PROGRAM MAIN
VAR	
	generateRecipe : BOOL;
	
	addRecipeToDB : AddRecipeToDatabase;
	validator : Validation;
	arrayHelpers : ArrayFunctions;
	
	resetAddRecipeToDatabase : AddRecipeToDatabase;
	resetValidation : Validation;
	resetArrayFunctions : ArrayFunctions;
	
	start : BOOL := TRUE;
END_VAR

validator(); //real time error/warning message generator

IF generateRecipe THEN
	addRecipeToDB();
	
	IF addRecipeToDB.finished THEN
		reset();
		//reset all variables
		generateRecipe := FALSE;
		RETURN;
	END_IF
END_IF

METHOD reset : BOOL
VAR_INPUT
END_VAR
//reset FBs
MEMCPY(ADR(addRecipeToDB), ADR(resetAddRecipeToDatabase), SIZEOF(AddRecipeToDatabase));
MEMCPY(ADR(validator), ADR(resetValidation), SIZEOF(Validation));
MEMCPY(ADR(arrayHelpers), ADR(resetArrayFunctions), SIZEOF(ArrayFunctions));

//reset fields
BundleData.id := '';
BundleData.weight := 0;
BundleData.length := 0;
BundleData.height := 0;
BundleData.width := 0;
BundleData.pieces := 0;
BundleData.layers := 0;
BundleData.piecesPerLayer := 0;
MEMSET(ADR(BundleData.requiredProcessing), 0, SIZEOF(BundleData.requiredProcessing));

ExtrusionData.extrusionWeight := 0;
ExtrusionData.extrusionHeight := 0;
ExtrusionData.extrusionWidth := 0;

MEMSET(ADR(StrapWrapRecipe.facePaper), 0, SIZEOF(StrapWrapRecipe.facePaper));
MEMSET(ADR(StrapWrapRecipe.faceCardboard), 0, SIZEOF(StrapWrapRecipe.faceCardboard));
MEMSET(ADR(StrapWrapRecipe.TopPaper), 0, SIZEOF(StrapWrapRecipe.TopPaper));
MEMSET(ADR(StrapWrapRecipe.LeftPaper), 0, SIZEOF(StrapWrapRecipe.LeftPaper));
MEMSET(ADR(StrapWrapRecipe.RightPaper), 0, SIZEOF(StrapWrapRecipe.RightPaper));
MEMSET(ADR(StrapWrapRecipe.BottomPaper), 0, SIZEOF(StrapWrapRecipe.BottomPaper));
MEMSET(ADR(StrapWrapRecipe.Cardboard), 0, SIZEOF(StrapWrapRecipe.Cardboard));
MEMSET(ADR(StrapWrapRecipe.CornerGuard), 0, SIZEOF(StrapWrapRecipe.CornerGuard));
MEMSET(ADR(StrapWrapRecipe.Chipboard), 0, SIZEOF(StrapWrapRecipe.Chipboard));
MEMSET(ADR(StrapWrapRecipe.WoodBunk), 0, SIZEOF(StrapWrapRecipe.WoodBunk));
END_METHOD

END_PROGRAM

(* stored: Version 1.1.0.1, ProductVersion 3.1.4024.11
   POU MAIN: Id {ff564e74-949a-4b82-bef1-798dfdd3f140}, SpecialFunc None
   Method reset: Id {f3587a12-2501-4871-ad4b-2c8e5ae64883} *)
